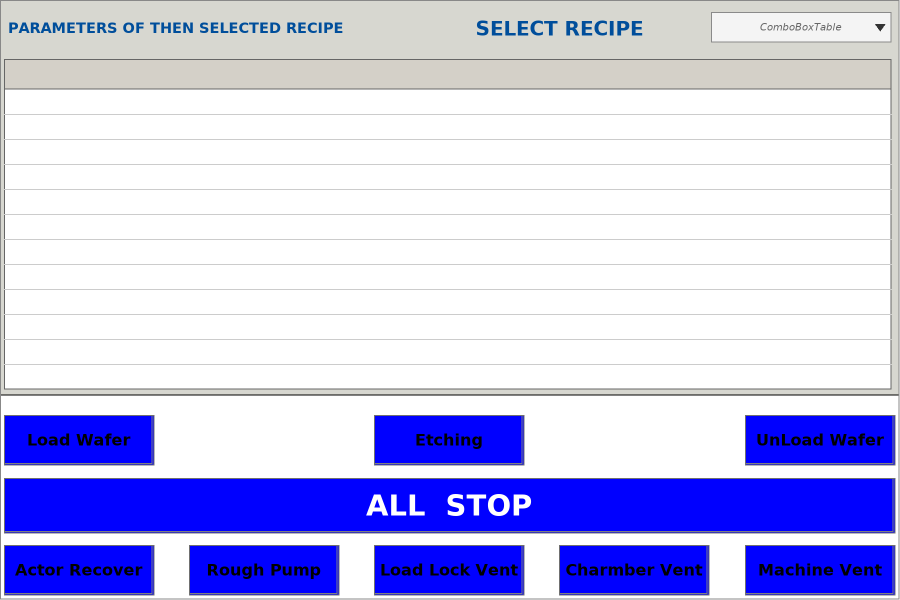
VISUALIZATION Recipe_Operator  // 900x600
    Rectangle (0,0 899x395)
    Table (4,59 887x330), data array: gRecipeViewData
        p1128707560: gShowNum
        p3854506369: gRecipeViewData[INDEX].NUM
        p1892666644: gRecipeViewData[INDEX].etchTime
        p338671338: gRecipeViewData[INDEX].rfPoint_Source
        p2170511999: gRecipeViewData[INDEX].pdvPoint
        p3723444502: gRecipeViewData[INDEX].mfc1
        p1218418051: gRecipeViewData[INDEX].mfc2
        p746581629: gRecipeViewData[INDEX].mfc3
        p3104783080: gRecipeViewData[INDEX].mfc4
        p2501879983: gRecipeViewData[INDEX].mfc5
        p7306298: gRecipeViewData[INDEX].mfc6
        p1933151965: gRecipeViewData[INDEX].mfc7
        p3863566920: gRecipeViewData[INDEX].mfc8
        p2192122294: gRecipeViewData[INDEX].mfc9
        p400160035: gRecipeViewData[INDEX].rfPoint_Power
        p1265227338: gRecipeViewData[INDEX].par_2
        p3726181087: gRecipeViewData[INDEX].par_3
        p3136911649: gRecipeViewData[INDEX].par_4
        p2237128397: N2(50)
        p505689113: CF4(200)
        p1757482276: CHF3(200)
        p4088588272: SF6(200)
        p2243050616: O2(100)
        p516019884: O2(10)
        p1739542657: He(500)
        p4242324053: Ar(500)
        p2319025000: C4F8(200)
        p3312258591: gRecipeViewData[INDEX].par1
        p1791247317: gRecipeViewData[INDEX].par2
        p262371475: gRecipeViewData[INDEX].par3
        p4008173056: gRecipeViewData[INDEX].par4
        p2340480326: gRecipeViewData[INDEX].par5
        p606709900: gRecipeViewData[INDEX].par6
        p1095668682: gRecipeViewData[INDEX].par7
        p1037165547: gRecipeViewData[INDEX].par8
        p1488378029: gRecipeViewData[INDEX].par9
        p152217274: gRecipeViewData[INDEX].par10
        p1819647484: gRecipeViewData[INDEX].par11
        p3286028342: gRecipeViewData[INDEX].par12
        p2797333360: gRecipeViewData[INDEX].par13
        p1207913955: gRecipeViewData[INDEX].par14
        p580417189: gRecipeViewData[INDEX].par15
        p2368813935: gRecipeViewData[INDEX].par16
    Rectangle (5,8 389x40), "PARAMETERS OF THEN SELECTED RECIPE"
    ComboBoxTable (711,12 180x30), variable: gRecipeSelectIndex1, data array: gRecipeNameSelect
        p1128707560: gRecipeSelctMaxIndex
        p3854506369: gRecipeNameSelect[INDEX].Name
    Rectangle (446,4 227x49), "SELECT RECIPE"
    Button (4,545 150x50), "Actor Recover", input disabled if: gSPOUBusy
        OnMouseClick: execute { S_ActuatorRecoveryPOU.Act_Init_Status(); S_ActuatorRecoveryPOU.Act_Ex(); }
    Button (189,545 150x50), "Rough Pump", input disabled if: gSPOUBusy
        OnMouseClick: execute { S_RoughPumping.Act_Init_Status(); S_RoughPumping.Act_Ex(); }
    Button (559,545 150x50), "Charmber Vent", input disabled if: gSPOUBusy
        OnMouseClick: execute { S_ChamberLLVent.Act_Init_Status(); S_ChamberLLVent.Act_Ex(); }
    Button (374,415 150x50), "Etching", input disabled if: gSPOUBusy
        OnMouseClick: execute { S_Etching.Act_Init_Status(); S_Etching.Act_Ex(); }
    Button (374,545 150x50), "Load Lock Vent", input disabled if: gSPOUBusy
        OnMouseClick: execute { S_LoadLockVent.Act_Init_Status(); S_LoadLockVent.Act_Ex(); }
    Button (4,415 150x50), "Load Wafer", input disabled if: gSPOUBusy
        OnMouseClick: execute { S_LoadWafer.Act_Init_Status(); S_LoadWafer.Act_Ex(); }
    Button (745,545 150x50), "Machine Vent", input disabled if: gSPOUBusy
        OnMouseClick: execute { S_MachineVent.Act_Init_Status(); S_MachineVent.Act_Ex(); }
    Button (745,415 150x50), "UnLoad Wafer", input disabled if: gSPOUBusy
        OnMouseClick: execute { S_UnLoadWafer.Act_Init_Status(); S_UnLoadWafer.Act_Ex(); }
    Button (4,478 891x55), "ALL STOP"
        tap MainRunPOU.AllAbort
        OnMouseClick: execute {
            gCtrlMode:=ControlMode.eManualCtrMode;
            IF RunningStatus.eErrorState<>gRunningState THEN
            	gRunningState:=RunningStatus.eManualState;
            END_IF
        }
END_VISUALIZATION

(* stored: Version 1.1.0.1, ProductVersion 3.1.4024.4
   Visu Recipe_Operator: Id {345690ef-470c-48ba-99f4-bf79d6328017} *)
